// TIA Portal V16 export
// export: Created 2023-03-29T11:03:21.5219756Z, ExportSetting WithDefaults, DisplayName Totally Integrated Automation Portal, DisplayVersion V16 Update 6, DisplayName TIA Portal Version Control Interface, DisplayVersion V16 Update 2, DisplayName TIA Portal Openness, DisplayVersion V16 Update 6, DisplayName STEP 7 Professional, DisplayVersion V16 Update 6, DisplayName STEP 7 Safety, DisplayVersion V16, DisplayName WinCC Advanced, DisplayVersion V16 Update 6
FUNCTION "Konwerter zegarów" : Void   // FC19, LAD
TITLE = Konwersja DTL na Real
{ S7_Optimized_Access := 'TRUE' }
AUTHOR : rtecmer
VERSION : 0.1
// Funkcja konwersji czasu na wartość liczbowa
// stored: AutoNumber true, IsIECCheckEnabled false, SetENOAutomatically false, UDAEnableTagReadback false
   VAR_INPUT
      isPumping : Bool;   // sygnał ustawione przetłaczanie
      isRecharging : Bool;   // sygnał ustawione dosianie
      isAutpumping : Bool;   // sygnał usawione automatyczne sterowanie
   END_VAR
   VAR_TEMP
      timePumpingOn : Real;   // czas start przetłaczanie
      timePumpingOff : Real;   // czas stop przetłaczanie
      timeRechargingOn : Real;   // czas strat dosilanie
      timeRechargingoff : Real;   // czas stop dosilanie
   END_VAR
BEGIN

REGION Network 1: RTC local
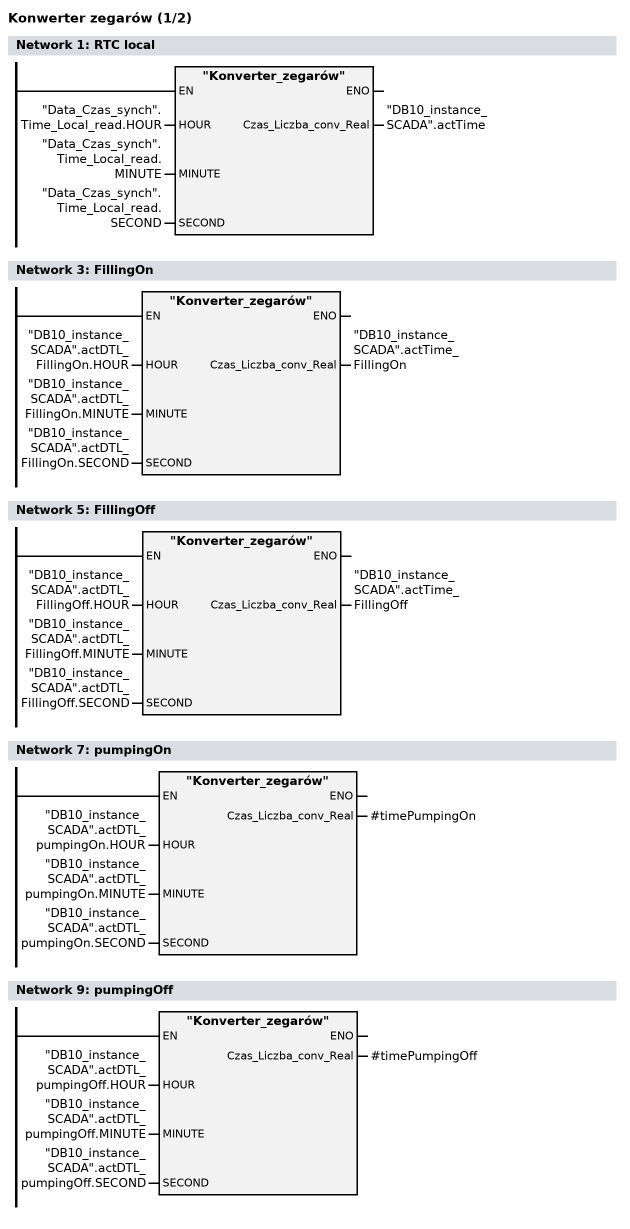
   RUNG wire#powerrail
      "Konverter_zegarów"(HOUR := "Data_Czas_synch".Time_Local_read.HOUR, MINUTE := "Data_Czas_synch".Time_Local_read.MINUTE, SECOND := "Data_Czas_synch".Time_Local_read.SECOND, Czas_Liczba_conv_Real => "DB10_instance_SCADA".actTime)
   END_RUNG
   // the same network as SCL:
   "Konverter_zegarów"(HOUR := "Data_Czas_synch".Time_Local_read.HOUR,
                       MINUTE := "Data_Czas_synch".Time_Local_read.MINUTE,
                       SECOND := "Data_Czas_synch".Time_Local_read.SECOND,
                       Czas_Liczba_conv_Real => "DB10_instance_SCADA".actTime);
END_REGION

REGION Network 3: FillingOn
   RUNG wire#powerrail
      "Konverter_zegarów"(HOUR := "DB10_instance_SCADA".actDTL_FillingOn.HOUR, MINUTE := "DB10_instance_SCADA".actDTL_FillingOn.MINUTE, SECOND := "DB10_instance_SCADA".actDTL_FillingOn.SECOND, Czas_Liczba_conv_Real => "DB10_instance_SCADA".actTime_FillingOn)
   END_RUNG
   // the same network as SCL:
   "Konverter_zegarów"(HOUR := "DB10_instance_SCADA".actDTL_FillingOn.HOUR,
                       MINUTE := "DB10_instance_SCADA".actDTL_FillingOn.MINUTE,
                       SECOND := "DB10_instance_SCADA".actDTL_FillingOn.SECOND,
                       Czas_Liczba_conv_Real => "DB10_instance_SCADA".actTime_FillingOn);
END_REGION

REGION Network 5: FillingOff
   RUNG wire#powerrail
      "Konverter_zegarów"(HOUR := "DB10_instance_SCADA".actDTL_FillingOff.HOUR, MINUTE := "DB10_instance_SCADA".actDTL_FillingOff.MINUTE, SECOND := "DB10_instance_SCADA".actDTL_FillingOff.SECOND, Czas_Liczba_conv_Real => "DB10_instance_SCADA".actTime_FillingOff)
   END_RUNG
   // the same network as SCL:
   "Konverter_zegarów"(HOUR := "DB10_instance_SCADA".actDTL_FillingOff.HOUR,
                       MINUTE := "DB10_instance_SCADA".actDTL_FillingOff.MINUTE,
                       SECOND := "DB10_instance_SCADA".actDTL_FillingOff.SECOND,
                       Czas_Liczba_conv_Real => "DB10_instance_SCADA".actTime_FillingOff);
END_REGION

REGION Network 7: pumpingOn
   RUNG wire#powerrail
      "Konverter_zegarów"(HOUR := "DB10_instance_SCADA".actDTL_pumpingOn.HOUR, MINUTE := "DB10_instance_SCADA".actDTL_pumpingOn.MINUTE, SECOND := "DB10_instance_SCADA".actDTL_pumpingOn.SECOND, Czas_Liczba_conv_Real => #timePumpingOn)
   END_RUNG
   // the same network as SCL:
   "Konverter_zegarów"(HOUR := "DB10_instance_SCADA".actDTL_pumpingOn.HOUR,
                       MINUTE := "DB10_instance_SCADA".actDTL_pumpingOn.MINUTE,
                       SECOND := "DB10_instance_SCADA".actDTL_pumpingOn.SECOND,
                       Czas_Liczba_conv_Real => #timePumpingOn);
END_REGION

REGION Network 9: pumpingOff
   RUNG wire#powerrail
      "Konverter_zegarów"(HOUR := "DB10_instance_SCADA".actDTL_pumpingOff.HOUR, MINUTE := "DB10_instance_SCADA".actDTL_pumpingOff.MINUTE, SECOND := "DB10_instance_SCADA".actDTL_pumpingOff.SECOND, Czas_Liczba_conv_Real => #timePumpingOff)
   END_RUNG
   // the same network as SCL:
   "Konverter_zegarów"(HOUR := "DB10_instance_SCADA".actDTL_pumpingOff.HOUR,
                       MINUTE := "DB10_instance_SCADA".actDTL_pumpingOff.MINUTE,
                       SECOND := "DB10_instance_SCADA".actDTL_pumpingOff.SECOND,
                       Czas_Liczba_conv_Real => #timePumpingOff);
END_REGION

REGION Network 11: RechargingOn
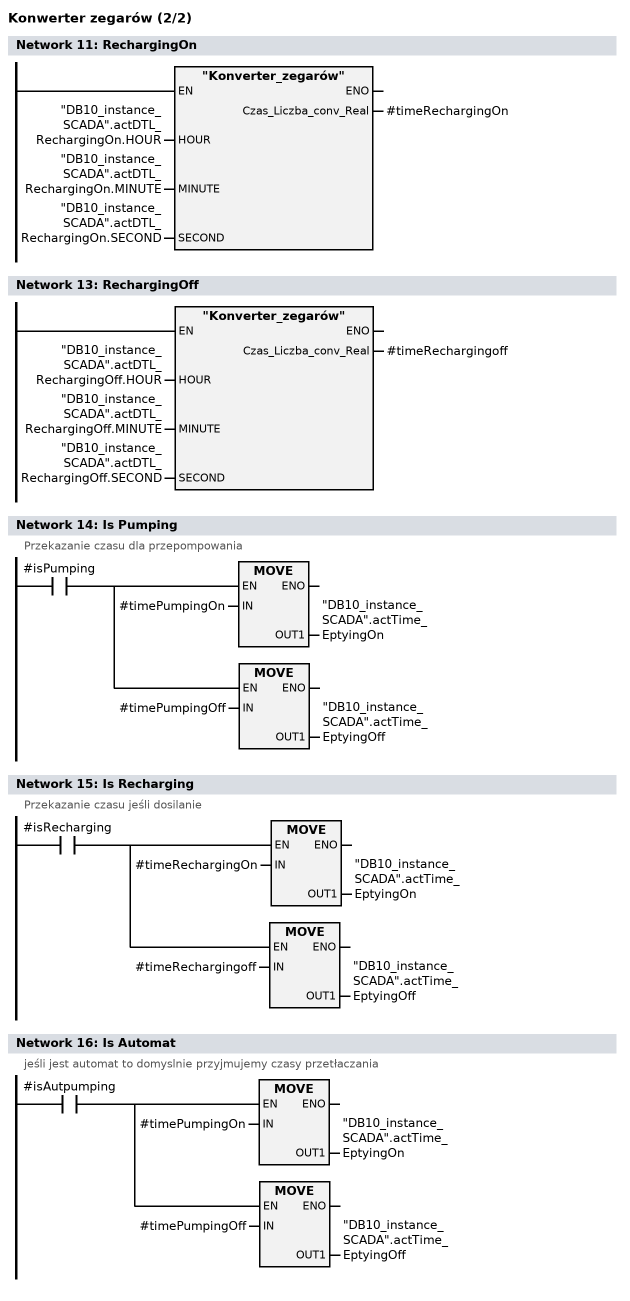
   RUNG wire#powerrail
      "Konverter_zegarów"(HOUR := "DB10_instance_SCADA".actDTL_RechargingOn.HOUR, MINUTE := "DB10_instance_SCADA".actDTL_RechargingOn.MINUTE, SECOND := "DB10_instance_SCADA".actDTL_RechargingOn.SECOND, Czas_Liczba_conv_Real => #timeRechargingOn)
   END_RUNG
   // the same network as SCL:
   "Konverter_zegarów"(HOUR := "DB10_instance_SCADA".actDTL_RechargingOn.HOUR,
                       MINUTE := "DB10_instance_SCADA".actDTL_RechargingOn.MINUTE,
                       SECOND := "DB10_instance_SCADA".actDTL_RechargingOn.SECOND,
                       Czas_Liczba_conv_Real => #timeRechargingOn);
END_REGION

REGION Network 13: RechargingOff
   RUNG wire#powerrail
      "Konverter_zegarów"(HOUR := "DB10_instance_SCADA".actDTL_RechargingOff.HOUR, MINUTE := "DB10_instance_SCADA".actDTL_RechargingOff.MINUTE, SECOND := "DB10_instance_SCADA".actDTL_RechargingOff.SECOND, Czas_Liczba_conv_Real => #timeRechargingoff)
   END_RUNG
   // the same network as SCL:
   "Konverter_zegarów"(HOUR := "DB10_instance_SCADA".actDTL_RechargingOff.HOUR,
                       MINUTE := "DB10_instance_SCADA".actDTL_RechargingOff.MINUTE,
                       SECOND := "DB10_instance_SCADA".actDTL_RechargingOff.SECOND,
                       Czas_Liczba_conv_Real => #timeRechargingoff);
END_REGION

REGION Network 14: Is Pumping
   // Przekazanie czasu dla przepompowania
   RUNG wire#powerrail
      Contact( #isPumping )
      wire#w1
      Move(in := #timePumpingOn, out1 => "DB10_instance_SCADA".actTime_EptyingOn)
   END_RUNG
   RUNG wire#w1
      Move(in := #timePumpingOff, out1 => "DB10_instance_SCADA".actTime_EptyingOff)
   END_RUNG
   // the same network as SCL:
   IF #isPumping THEN
       "DB10_instance_SCADA".actTime_EptyingOn := #timePumpingOn;
       "DB10_instance_SCADA".actTime_EptyingOff := #timePumpingOff;
   END_IF;
END_REGION

REGION Network 15: Is Recharging
   // Przekazanie czasu jeśli dosilanie
   RUNG wire#powerrail
      Contact( #isRecharging )
      wire#w1
      Move(in := #timeRechargingOn, out1 => "DB10_instance_SCADA".actTime_EptyingOn)
   END_RUNG
   RUNG wire#w1
      Move(in := #timeRechargingoff, out1 => "DB10_instance_SCADA".actTime_EptyingOff)
   END_RUNG
   // the same network as SCL:
   IF #isRecharging THEN
       "DB10_instance_SCADA".actTime_EptyingOn := #timeRechargingOn;
       "DB10_instance_SCADA".actTime_EptyingOff := #timeRechargingoff;
   END_IF;
END_REGION

REGION Network 16: Is Automat
   // jeśli jest automat to domyslnie przyjmujemy czasy przetłaczania
   RUNG wire#powerrail
      Contact( #isAutpumping )
      wire#w1
      Move(in := #timePumpingOn, out1 => "DB10_instance_SCADA".actTime_EptyingOn)
   END_RUNG
   RUNG wire#w1
      Move(in := #timePumpingOff, out1 => "DB10_instance_SCADA".actTime_EptyingOff)
   END_RUNG
   // the same network as SCL:
   IF #isAutpumping THEN
       "DB10_instance_SCADA".actTime_EptyingOn := #timePumpingOn;
       "DB10_instance_SCADA".actTime_EptyingOff := #timePumpingOff;
   END_IF;
END_REGION
END_FUNCTION
